FUNCTION_BLOCK fbBrensonMultiFreqCtrl
VAR_INPUT

	bErrorReset : BOOL;
	b2550NewFirmware : BOOL;
END_VAR

VAR_IN_OUT PERSISTENT
	DSBrensonGenerator : ARRAY [1..iUSGeneratorQty] OF DS_BrensonGenerator;
	iStepDelaySVns: INT;
END_VAR

VAR_OUTPUT
	bFSel1OnOff :  BOOL;
	bFSel2OnOff :  BOOL;

END_VAR

VAR PERSISTENT
	ARbFreqChangeTriggerEn : ARRAY [1..iUSGeneratorQty] OF BOOL; (*Internally activate by monitor the changes of set point*)
(*	ARiPowerAnalogInput AT %I* : ARRAY [1..iUSGeneratorQty] OF INT; (*Link to Terminal*)
	ARiPowerAnalogOutput AT %Q* : ARRAY [1..iUSGeneratorQty] OF INT; (*Link to Terminal*)
*)
(**)	bFreqSwitchingPBRE: ARRAY [1..iUSGeneratorQty] OF R_TRIG;
	ARbFreqChangeMonitoringEn : ARRAY [1..iUSGeneratorQty] OF BOOL; (*Enable monitor the changes of set point*)
	ARiCurrentFreq: ARRAY [1..iUSGeneratorQty] OF INT;
	iFreqChangeStep: INT;
	iFreqChangeTriggerSet: INT;
	ARbFreqChangeTriggerEnRE: ARRAY [1..iUSGeneratorQty] OF R_TRIG;
	tStep1DelayTimer: TON;
	tStep2DelayTimer: TON;
	tStep3DelayTimer: TON;
	tStep0DelayTimer: TON;
	iGenFL: INT;
	iFreqChangeFL: INT;
END_VAR

(*Ultrasonic Start/Stop Ctrl*)
tStep0DelayTimer(IN:=iFreqChangeStep = 0 , PT:=INT_TO_TIME(iStepDelaySVns) , Q=> , ET=> );

iGenFL := 1;

	FOR iGenFL := 1 TO iUSGeneratorQty DO

				(*Min Control - Default*)
				IF DSBrensonGenerator[iGenFL].IN_lrPowerToAnalogRatio <= 0 THEN
				DSBrensonGenerator[iGenFL].IN_lrPowerToAnalogRatio := 327.67;
				END_IF

				(*Ultrasonic Start/Stop Ctrl*)
				IF tStep0DelayTimer.Q THEN
					IF DSBrensonGenerator[iGenFL].IN_bUltrasonicStartEn THEN
					DSBrensonGenerator[iGenFL].OUT_bUltrasonicOnOff := TRUE;
					ELSE
					DSBrensonGenerator[iGenFL].OUT_bUltrasonicOnOff := FALSE;
					END_IF

				END_IF


				(*MultiFreq Ctrl - Change Freq via Digital Output Control*)

				(*Monitoring Start/Stop Control*)
				IF DSBrensonGenerator[iGenFL].IN_bMultiFreqEn THEN
					IF DSBrensonGenerator[iGenFL].DSBrensonMulFreqSwitching.bFreqRange2550En AND NOT DSBrensonGenerator[iGenFL].DSBrensonMulFreqSwitching.bFreqRange4080120En THEN
						IF DSBrensonGenerator[iGenFL].IN_iFreqSetPoint = 25 OR DSBrensonGenerator[iGenFL].IN_iFreqSetPoint = 50 THEN
						ARbFreqChangeMonitoringEn[iGenFL] := TRUE;
						END_IF
					ELSIF NOT DSBrensonGenerator[iGenFL].DSBrensonMulFreqSwitching.bFreqRange2550En AND DSBrensonGenerator[iGenFL].DSBrensonMulFreqSwitching.bFreqRange4080120En THEN
						IF DSBrensonGenerator[iGenFL].IN_iFreqSetPoint = 40 OR DSBrensonGenerator[iGenFL].IN_iFreqSetPoint = 80 OR DSBrensonGenerator[iGenFL].IN_iFreqSetPoint = 120 THEN
						ARbFreqChangeMonitoringEn[iGenFL] := TRUE;
						END_IF
					ELSE
						ARbFreqChangeMonitoringEn[iGenFL] := FALSE;
					END_IF
				ELSE
						ARbFreqChangeMonitoringEn[iGenFL] := FALSE;
				END_IF

				IF ARbFreqChangeMonitoringEn[iGenFL] THEN

					IF DSBrensonGenerator[iGenFL].IN_iFreqSetPoint <> ARiCurrentFreq[iGenFL] THEN
						ARbFreqChangeTriggerEn[iGenFL] := TRUE;
					END_IF

				ELSE
					ARbFreqChangeTriggerEn[iGenFL] := FALSE;
				END_IF


				(*Analog Output*)
				IF DSBrensonGenerator[iGenFL].IN_lrAnalogOutputFineTuneRatio <= 0 THEN
				DSBrensonGenerator[iGenFL].IN_lrAnalogOutputFineTuneRatio := 1;
				END_IF

				IF DSBrensonGenerator[iGenFL].IN_iTargetPowerPercentSetPoint <= 0 THEN
				DSBrensonGenerator[iGenFL].OUT_iPowerAnalogOutput := 0;
				ELSIF DSBrensonGenerator[iGenFL].IN_lrPowerToAnalogRatio <= 0 THEN
				DSBrensonGenerator[iGenFL].OUT_iPowerAnalogOutput := 0;
				ELSIF (INT_TO_LREAL(DSBrensonGenerator[iGenFL].IN_iTargetPowerPercentSetPoint) * DSBrensonGenerator[iGenFL].IN_lrPowerToAnalogRatio) * DSBrensonGenerator[iGenFL].IN_lrAnalogOutputFineTuneRatio <=32767 THEN
					DSBrensonGenerator[iGenFL].OUT_iPowerAnalogOutput := LREAL_TO_INT(INT_TO_LREAL(DSBrensonGenerator[iGenFL].IN_iTargetPowerPercentSetPoint) * DSBrensonGenerator[iGenFL].IN_lrPowerToAnalogRatio * DSBrensonGenerator[iGenFL].IN_lrAnalogOutputFineTuneRatio);
				ELSIF (INT_TO_LREAL(DSBrensonGenerator[iGenFL].IN_iTargetPowerPercentSetPoint) * DSBrensonGenerator[iGenFL].IN_lrPowerToAnalogRatio * DSBrensonGenerator[iGenFL].IN_lrAnalogOutputFineTuneRatio) >32767 THEN
					DSBrensonGenerator[iGenFL].OUT_iPowerAnalogOutput := 32767;

				ELSE
				DSBrensonGenerator[iGenFL].OUT_iPowerAnalogOutput := 0;
				END_IF


				(*ActualPowerPercentageDisplay*)

				IF DSBrensonGenerator[iGenFL].IN_lrAnalogInputFineTuneRatio <= 0 THEN
				DSBrensonGenerator[iGenFL].IN_lrAnalogInputFineTuneRatio := 1;
				END_IF

				IF DSBrensonGenerator[iGenFL].IN_iPowerAnalogInput <= 0 THEN
				DSBrensonGenerator[iGenFL].OUT_iActualPowerPercentDisplay := 0;
				ELSIF DSBrensonGenerator[iGenFL].IN_lrPowerToAnalogRatio <= 0 THEN
				DSBrensonGenerator[iGenFL].OUT_iActualPowerPercentDisplay := 0;
				ELSIF ((INT_TO_LREAL(DSBrensonGenerator[iGenFL].IN_iPowerAnalogInput) / DSBrensonGenerator[iGenFL].IN_lrPowerToAnalogRatio) )* DSBrensonGenerator[iGenFL].IN_lrAnalogInputFineTuneRatio <=100 THEN
					DSBrensonGenerator[iGenFL].OUT_iActualPowerPercentDisplay := LREAL_TO_INT((INT_TO_LREAL(DSBrensonGenerator[iGenFL].IN_iPowerAnalogInput) / DSBrensonGenerator[iGenFL].IN_lrPowerToAnalogRatio) * DSBrensonGenerator[iGenFL].IN_lrAnalogInputFineTuneRatio);
				ELSIF ((INT_TO_LREAL(DSBrensonGenerator[iGenFL].IN_iPowerAnalogInput) / DSBrensonGenerator[iGenFL].IN_lrPowerToAnalogRatio) )* DSBrensonGenerator[iGenFL].IN_lrAnalogInputFineTuneRatio >100 THEN
					DSBrensonGenerator[iGenFL].OUT_iActualPowerPercentDisplay := 100;

				ELSE
				DSBrensonGenerator[iGenFL].OUT_iPowerAnalogOutput := 0;
				END_IF

				(*TS - FreqSwitchingPushButtonControl*)
				bFreqSwitchingPBRE[iGenFL](CLK:=DSBrensonGenerator[iGenFL].DSBrensonMulFreqSwitching.bFreqSwitchingPB_TS , Q=> );

				IF NOT DSBrensonGenerator[iGenFL].DSBrensonMulFreqSwitching.bFreqRange2550En AND NOT DSBrensonGenerator[iGenFL].DSBrensonMulFreqSwitching.bFreqRange4080120En THEN
				DSBrensonGenerator[iGenFL].DSBrensonMulFreqSwitching.iFreqOutput_TS := 0;
				ELSIF DSBrensonGenerator[iGenFL].DSBrensonMulFreqSwitching.bFreqRange2550En AND DSBrensonGenerator[iGenFL].DSBrensonMulFreqSwitching.bFreqRange4080120En THEN
				DSBrensonGenerator[iGenFL].DSBrensonMulFreqSwitching.iFreqOutput_TS := 0;


				ELSIF DSBrensonGenerator[iGenFL].DSBrensonMulFreqSwitching.bFreqRange2550En AND NOT DSBrensonGenerator[iGenFL].DSBrensonMulFreqSwitching.bFreqRange4080120En THEN

					IF DSBrensonGenerator[iGenFL].DSBrensonMulFreqSwitching.iFreqOutput_TS <> 25 AND DSBrensonGenerator[iGenFL].DSBrensonMulFreqSwitching.iFreqOutput_TS <> 50 THEN
					DSBrensonGenerator[iGenFL].DSBrensonMulFreqSwitching.iFreqOutput_TS := 25;
					END_IF

					IF bFreqSwitchingPBRE[iGenFL].Q THEN
						IF DSBrensonGenerator[iGenFL].DSBrensonMulFreqSwitching.iFreqOutput_TS = 25 THEN
						DSBrensonGenerator[iGenFL].DSBrensonMulFreqSwitching.iFreqOutput_TS := 50;
						ELSIF DSBrensonGenerator[iGenFL].DSBrensonMulFreqSwitching.iFreqOutput_TS = 50 THEN
						DSBrensonGenerator[iGenFL].DSBrensonMulFreqSwitching.iFreqOutput_TS := 25;
						END_IF
					END_IF


				ELSIF NOT DSBrensonGenerator[iGenFL].DSBrensonMulFreqSwitching.bFreqRange2550En AND DSBrensonGenerator[iGenFL].DSBrensonMulFreqSwitching.bFreqRange4080120En THEN

					IF DSBrensonGenerator[iGenFL].DSBrensonMulFreqSwitching.iFreqOutput_TS <> 40 AND DSBrensonGenerator[iGenFL].DSBrensonMulFreqSwitching.iFreqOutput_TS <> 80 AND DSBrensonGenerator[iGenFL].DSBrensonMulFreqSwitching.iFreqOutput_TS <> 120  THEN
					DSBrensonGenerator[iGenFL].DSBrensonMulFreqSwitching.iFreqOutput_TS := 40;
					END_IF

					IF bFreqSwitchingPBRE[iGenFL].Q AND NOT DSBrensonGenerator[iGenFL].DSBrensonMulFreqSwitching.bDisableMultiFreq80kHz THEN
						IF DSBrensonGenerator[iGenFL].DSBrensonMulFreqSwitching.iFreqOutput_TS = 40 THEN
						DSBrensonGenerator[iGenFL].DSBrensonMulFreqSwitching.iFreqOutput_TS := 80;
						ELSIF DSBrensonGenerator[iGenFL].DSBrensonMulFreqSwitching.iFreqOutput_TS = 80 THEN
						DSBrensonGenerator[iGenFL].DSBrensonMulFreqSwitching.iFreqOutput_TS := 120;
						ELSIF DSBrensonGenerator[iGenFL].DSBrensonMulFreqSwitching.iFreqOutput_TS = 120 THEN
						DSBrensonGenerator[iGenFL].DSBrensonMulFreqSwitching.iFreqOutput_TS := 40;
						END_IF

					ELSIF bFreqSwitchingPBRE[iGenFL].Q AND DSBrensonGenerator[iGenFL].DSBrensonMulFreqSwitching.bDisableMultiFreq80kHz THEN
						IF DSBrensonGenerator[iGenFL].DSBrensonMulFreqSwitching.iFreqOutput_TS = 40 THEN
						DSBrensonGenerator[iGenFL].DSBrensonMulFreqSwitching.iFreqOutput_TS := 120;
						ELSIF DSBrensonGenerator[iGenFL].DSBrensonMulFreqSwitching.iFreqOutput_TS = 120 THEN
						DSBrensonGenerator[iGenFL].DSBrensonMulFreqSwitching.iFreqOutput_TS := 40;
						END_IF

					END_IF

				END_IF

	END_FOR



(*Seperate FL to control*)

IF iFreqChangeStep = 0 THEN
iFreqChangeFL := 1;
	FOR iFreqChangeFL := 1 TO iUSGeneratorQty DO

		IF ARbFreqChangeTriggerEn[iFreqChangeFL] THEN
		iFreqChangeStep := 1;
		iFreqChangeTriggerSet := iFreqChangeFL;
		iFreqChangeFL := iUSGeneratorQty +1;
		END_IF
	END_FOR
END_IF

(*******************************************************************************************)






(*Freq Change Start*)

IF iStepDelaySVns < 300 THEN
iStepDelaySVns := 300;
END_IF


(*Freq Change Sequence Start*)
tStep1DelayTimer(IN:=iFreqChangeStep=1 , PT:=INT_TO_TIME(iStepDelaySVns) , Q=> , ET=> );
tStep2DelayTimer(IN:=iFreqChangeStep=2 , PT:=INT_TO_TIME(iStepDelaySVns) , Q=> , ET=> );
tStep3DelayTimer(IN:=iFreqChangeStep=3 , PT:=INT_TO_TIME(iStepDelaySVns) , Q=> , ET=> );

CASE iFreqChangeStep OF
0:
	bFSel1OnOff := FALSE;
	bFSel2OnOff := FALSE;


1:
DSBrensonGenerator[iFreqChangeTriggerSet].OUT_bUltrasonicOnOff := FALSE;

IF DSBrensonGenerator[iFreqChangeTriggerSet].DSBrensonMulFreqSwitching.bFreqRange2550En AND NOT b2550NewFirmware THEN

	IF DSBrensonGenerator[iFreqChangeTriggerSet].IN_iFreqSetPoint = 25 THEN
	bFSel1OnOff := TRUE;
	bFSel2OnOff := FALSE;
	ELSIF DSBrensonGenerator[iFreqChangeTriggerSet].IN_iFreqSetPoint = 50 THEN
	bFSel1OnOff := FALSE;
	bFSel2OnOff := TRUE;
	ELSIF DSBrensonGenerator[iFreqChangeTriggerSet].IN_iFreqSetPoint = 0 THEN
	bFSel1OnOff := FALSE;
	bFSel2OnOff := FALSE;
	ELSE
	bFSel1OnOff := FALSE;
	bFSel2OnOff := FALSE;
	iFreqChangeStep := 4;
	END_IF

ELSIF DSBrensonGenerator[iFreqChangeTriggerSet].DSBrensonMulFreqSwitching.bFreqRange2550En AND b2550NewFirmware THEN

	IF DSBrensonGenerator[iFreqChangeTriggerSet].IN_iFreqSetPoint = 25 THEN
	bFSel1OnOff := TRUE;
	bFSel2OnOff := TRUE;
	ELSIF DSBrensonGenerator[iFreqChangeTriggerSet].IN_iFreqSetPoint = 50 THEN
	bFSel1OnOff := FALSE;
	bFSel2OnOff := TRUE;
	ELSIF DSBrensonGenerator[iFreqChangeTriggerSet].IN_iFreqSetPoint = 0 THEN
	bFSel1OnOff := FALSE;
	bFSel2OnOff := FALSE;
	ELSE
	bFSel1OnOff := FALSE;
	bFSel2OnOff := FALSE;
	iFreqChangeStep := 4;
	END_IF

END_IF

IF DSBrensonGenerator[iFreqChangeTriggerSet].DSBrensonMulFreqSwitching.bFreqRange4080120En THEN

	IF NOT DSBrensonGenerator[iFreqChangeTriggerSet].DSBrensonMulFreqSwitching.bDisableMultiFreq80kHz THEN

			IF DSBrensonGenerator[iFreqChangeTriggerSet].IN_iFreqSetPoint = 40 THEN
			bFSel1OnOff := TRUE;
			bFSel2OnOff := TRUE;
			ELSIF DSBrensonGenerator[iFreqChangeTriggerSet].IN_iFreqSetPoint = 80 THEN
			bFSel1OnOff := FALSE;
			bFSel2OnOff := TRUE;
			ELSIF DSBrensonGenerator[iFreqChangeTriggerSet].IN_iFreqSetPoint = 120 THEN
			bFSel1OnOff := TRUE;
			bFSel2OnOff := FALSE;
			ELSIF DSBrensonGenerator[iFreqChangeTriggerSet].IN_iFreqSetPoint = 0 THEN
			bFSel1OnOff := FALSE;
			bFSel2OnOff := FALSE;
			ELSE
			bFSel1OnOff := FALSE;
			bFSel2OnOff := FALSE;
			iFreqChangeStep := 4;
			END_IF
	ELSE

			IF DSBrensonGenerator[iFreqChangeTriggerSet].IN_iFreqSetPoint = 40 THEN
			bFSel1OnOff := TRUE;
			bFSel2OnOff := FALSE;
			ELSIF DSBrensonGenerator[iFreqChangeTriggerSet].IN_iFreqSetPoint = 120 THEN
			bFSel1OnOff := FALSE;
			bFSel2OnOff := TRUE;
			ELSIF DSBrensonGenerator[iFreqChangeTriggerSet].IN_iFreqSetPoint = 0 THEN
			bFSel1OnOff := FALSE;
			bFSel2OnOff := FALSE;
			ELSE
			bFSel1OnOff := FALSE;
			bFSel2OnOff := FALSE;
			iFreqChangeStep := 4;
			END_IF
	END_IF



END_IF


IF tStep1DelayTimer.Q THEN
iFreqChangeStep := 2;
END_IF

2:
IF DSBrensonGenerator[iFreqChangeTriggerSet].IN_iFreqSetPoint <> 0 THEN
DSBrensonGenerator[iFreqChangeTriggerSet].OUT_bUltrasonicOnOff := TRUE;
ELSE
DSBrensonGenerator[iFreqChangeTriggerSet].OUT_bUltrasonicOnOff := FALSE;
END_IF

IF tStep2DelayTimer.Q THEN
iFreqChangeStep := 3;
END_IF

3:
DSBrensonGenerator[iFreqChangeTriggerSet].OUT_bUltrasonicOnOff := FALSE;
bFSel1OnOff := FALSE;
bFSel2OnOff := FALSE;

IF tStep3DelayTimer.Q THEN
iFreqChangeStep := 0;
ARbFreqChangeTriggerEn[iFreqChangeTriggerSet] := FALSE;
ARiCurrentFreq[iFreqChangeTriggerSet] := DSBrensonGenerator[iFreqChangeTriggerSet].IN_iFreqSetPoint;
END_IF

4: (*Error*)
DSBrensonGenerator[iFreqChangeTriggerSet].OUT_bFreqSetPointError := TRUE;
iFreqChangeStep := 5;


5: (*Error - Waiting Reset*)
IF bErrorReset THEN
DSBrensonGenerator[iFreqChangeTriggerSet].OUT_bFreqSetPointError := FALSE;
iFreqChangeStep := 0;
ARbFreqChangeTriggerEn[iFreqChangeTriggerSet] := FALSE;
ARiCurrentFreq[iFreqChangeTriggerSet] := DSBrensonGenerator[iFreqChangeTriggerSet].IN_iFreqSetPoint;
END_IF

END_CASE

END_FUNCTION_BLOCK

(* stored: Version 1.1.0.1, ProductVersion 3.1.4024.12
   POU fbBrensonMultiFreqCtrl: Id {45a120e8-e921-4997-86d5-cdc8990417b9}, SpecialFunc None *)
